// TIA Portal V19 export
TYPE "LAF_typeVfdParameters"
// stored: Access Published
   STRUCT
      general : "LAF_typeVfdGeneralParameters";
      manual : "LAF_typeVfdMannualParameters";
      production : "LAF_typeVfdProductionParameters";
      maintenance { S7_SetPoint := 'True'} : "LAF_typeVfdMaintanceParameters";
   END_STRUCT;
END_TYPE
